{attribute 'qualified_only'}
VAR_GLOBAL PERSISTENT
	// Last valid incremental-axis coordinates. MAIN updates these only while
	// TwinCAT considers the corresponding NC axis referenced.
	fLastPositionX      : LREAL;
	fLastPositionY      : LREAL;
	bLastPositionValidX : BOOL;
	bLastPositionValidY : BOOL;
END_VAR

(* stored: Version 1.1.0.1, ProductVersion 3.1.4024.15
   GVL GVL_Persistent: Id {6c4627c9-22e3-4ac5-9eb9-b470f7393588} *)
